FUNCTION_BLOCK FB_MotionAxis_MC

VAR_INPUT
	ZSN	   			: BOOL												;
	ZSP				: BOOL												; 
	Exceeding_us			: INT;
	sNameAxis				: STRING [40];

END_VAR         	
                	
VAR  
	rtFirstCycle	: R_TRIG;						
	mcHomeAxis		: 	MC_HomeAxis						;//ADD BY EVAN 
	sAxisName		: STRING											;//Axis name          	
	xPlus			: BOOL												;	
	xMinus			: BOOL												;
	bDone			: BOOL												;	

// Variables for Hard Stop Homing	                        			
	iStatehsHomig	: E_HomingSteps := E_HomingSteps.IDLE				;
	rtHome			: R_TRIG											;
	rtHomeReset		: R_TRIG											;
	tonTimeOut		: TON												;
	xTimerStart		: BOOL												;
	bLSDefaultVal	: BOOL												; // Save Def value from driver
	xHomeError		: BOOL												;
// Variables for Force Control          					

	rtForceC		: R_TRIG											;
	rtForceCReset	: R_TRIG											;
	DelMaxPos		: LREAL 											;
	rCurrLimit		: LREAL												;
	StartPos		: LREAL												;
	xForceCError	: BOOL												;
//	Variables for Backlash Compensation
	rLastMove		: LREAL := 1										;
	tonBackComp		: TON												;
	rBacklashPer	: LREAL												;	
	
// Variables for errors
	rtError					:	R_TRIG;
	pTextType				:	POINTER TO STRING;
	sAxisErrorID			:	STRING(10);	
	ErrorMSG				:	STRING[255];

//	Exceeding time measuring
	sysTime					:	GETCPUCOUNTER;//GETSYSTEMTIME;					//	Used to measure execution time.
	uStartTime				:	UDINT;
	uFinishTime				:	UDINT;
	ftimeDiff				:	REAL;
	ton_dly	: TON;
	offset	: WORD;
END_VAR         	
                	
VAR_IN_OUT      	
	IN_OUT 			: ST_MotionAxis_MC	;//struct for each axis
	AXIS 			: AXIS_REF			;//Axis obj	
END_VAR

VAR_OUTPUT
	xError			: BOOL				;
	xBusy			: BOOL				;
END_VAR
VAR CONSTANT
	parallelGroupTLName		:	STRING := 'Port_851.TL_Axis_Error';
END_VAR

(* Power options ********************************************************************************************)			
IN_OUT.mcPower(
	Axis				:= AXIS, 
	Enable				:= , 
	Enable_Positive		:= ZSP, 
	Enable_Negative		:= ZSN OR IN_OUT.mcHome.Busy, 
	Override			:= , 
	BufferMode			:= , 
	Options				:= , 
	Status				=> , 
	Busy				=> , 
	Active				=> , 
	Error				=> , 
	ErrorID				=> );
	
(* Halt Mode ********************************************************************************************)	
IN_OUT.mcHalt(
	Axis				:= AXIS, 
	Execute				:= , 
	Deceleration		:= IN_OUT.rDeceleration, 
	Jerk				:= , 
	BufferMode			:= , 
	Options				:= , 
	Done				=> , 
	Busy				=> , 
	Active				=> , 
	CommandAborted		=> , 
	Error				=> , 
	ErrorID				=> );
	
(* Homing ***********************************************************************************************)
IN_OUT.mcHome(
	Axis				:= AXIS, 
	Execute				:= , 
	Position			:= in_out.rFirstpos, 
	HomingMode			:= MC_Direct, 
	BufferMode			:= , 
	Options				:= , 
	bCalibrationCam		:= ,//NOT  ZSN, 
	Done				=> , 
	Busy				=> , 
	Active				=> , 
	CommandAborted		=> , 
	Error				=> , 
	ErrorID				=> );
	
(* JOG **************************************************************************************************)
IN_OUT.mcJog(
	Axis				:= AXIS, 
	JogForward			:= , 
	JogBackwards		:= , 
	Mode				:= E_JogMode.MC_JOGMODE_CONTINOUS, 
	Position			:= , 
	Velocity			:= IN_OUT.rVelocity, 
	Acceleration		:= IN_OUT.rAcceleration, 
	Deceleration		:= IN_OUT.rDeceleration, 
	Jerk				:= IN_OUT.rJerk, 
	Done				=> , 
	Busy				=> , 
	Active				=> , 
	CommandAborted		=> , 
	Error				=> , 
	ErrorID				=> );
	
(* Move Absolute ****************************************************************************************)	
IN_OUT.mcMoveAbsolute(
	Axis				:= AXIS, 
	Execute				:= , 
	Position			:= IN_OUT.rActualPosSet, 
	Velocity			:= IN_OUT.rVelocitySet,     
	Acceleration		:= IN_OUT.rAcceleration, 
	Deceleration		:= IN_OUT.rDeceleration, 
	Jerk				:= IN_OUT.rJerk,         
	BufferMode			:= , 
	Options				:= , 
	Done				=> , 
	Busy				=> , 
	Active				=> , 
	CommandAborted		=> , 
	Error				=> , 
	ErrorID				=> );

	IF IN_OUT.bMoveAbsHMI THEN
		IN_OUT.mcMoveAbsolute.Execute	:= TRUE;
		IN_OUT.rActualPosSet	:= IN_OUT.rActualPosHMI;
		IN_OUT.rVelocitySet		:= IN_OUT.rVeloPers;
	END_IF
(* Move Relative *********************************************************************************************************)
IN_OUT.mcMoveRelative(
	Axis				:= AXIS, 
	Execute				:= , 
	Distance			:= IN_OUT.rPosition + IN_OUT.rBacklashvalue, 
	Velocity			:= IN_OUT.rVelocity,      
	Acceleration		:= IN_OUT.rAcceleration,  
	Deceleration		:= IN_OUT.rDeceleration,  
	Jerk				:= IN_OUT.rJerk,          
	BufferMode			:= ,
	Options				:= , 
	Done				=> bDone, 
	Busy				=> , 
	Active				=> , 
	CommandAborted		=> , 
	Error				=> , 
	ErrorID				=> );
	
(* Move Velocity *********************************************************************************************************)
	
IN_OUT.mcMoveVelocity(
	Axis				:=	AXIS,
	Execute				:=	,
	Velocity			:=	IN_OUT.rVelocity,
	Acceleration		:=	IN_OUT.rAcceleration,
	Deceleration		:=	IN_OUT.rDeceleration,
	Jerk				:=	IN_OUT.rJerk,
	Direction			:=	IN_OUT.axisDirection,
	BufferMode			:=	,
	Options				:=	,
	InVelocity			=>	,
	Busy				=>	,
	Active				=>	,
	CommandAborted		=>	,
	Error				=>	,
	ErrorID				=>	);
	
(**)	
IN_OUT.mcReadStatus(
	Axis				:= AXIS, 
	Enable				:= TRUE, 
	Valid				=> , 
	Busy				=> , 
	Error				=> , 
	ErrorID				=> , 
	ErrorStop			=> , 
	Disabled			=> , 
	Stopping			=> , 
	StandStill			=> , 
	DiscreteMotion		=> , 
	ContinuousMotion	=> , 
	SynchronizedMotion	=> , 
	Homing				=> , 
	ConstantVelocity	=> , 
	Accelerating		=> , 
	Decelerating		=> , 
	Status				=> );
	
(* Reset ************************************************************************************************)
IN_OUT.mcReset(
	Axis				:= AXIS, 
	Execute				:= , 
	Done				=> , 
	Busy				=> , 
	Error				=> , 
	ErrorID				=> );
	
(* Stop *************************************************************************************************)
IN_OUT.mcStop(
	Axis				:= AXIS, 
	Execute				:= , 
	Deceleration		:= , 
	Jerk				:= , 
	Options				:= , 
	Done				=> , 
	Busy				=> , 
	Active				=> , 
	CommandAborted		=> , 
	Error				=> , 
	ErrorID				=> );

(* Set Position *************************************************************************************************)
in_out.mcSetpoint(
	Axis			 := AXIS, 
	Execute			 := , 
	Position		 := IN_OUT.rSetPos, 
	Mode			 := , 
	Options			 := , 
	Done			 => , 
	Busy			 => , 
	Error			 => , 
	ErrorID			 => );


(* write status *************************************************************************************************)
IN_OUT.mcWriteBoolParameter(
	Axis			:= 	AXIS, 
	Execute:= 				, 
	ParameterNumber:= 		, 
	Value:= , 
	Done=> , 
	Busy=> , 
	Error=> , 
	ErrorID=> );

(* Read status *************************************************************************************************)
IN_OUT.mcReadBoolParameter(
	Axis:= AXIS, 
	Enable:= , 
	ParameterNumber:= , 
	ReadMode:= , 
	Valid=> , 
	Busy=> , 
	Error=> , 
	ErrorID=> , 
	Value=> );	

(*Read Actualposition***************************************************************)
IN_OUT.mcReadActualPosition(
	Axis:= AXIS, 
	Enable:= TRUE, 
	Valid=> , 
	Busy=> , 
	Error=> , 
	ErrorID=> , 
	Position=> IN_OUT.rActualPos );   
(*COE write**************************************************************************)	

IN_OUT.CoeWrt(
	sNetId:= IN_OUT.sNetID, 
	nSlaveAddr:= IN_OUT.nSlaveAddr, 
	nSubIndex:= IN_OUT.nSubIndex, 
	nIndex:= IN_OUT.nIndex, 
	pSrcBuf:= ADR(IN_OUT.iSdoWrite), 
	cbBufLen:= SIZEOF(IN_OUT.iSdoWrite), 
	bExecute:= , 
	tTimeout:= , 
	bBusy=> , 
	bError=> , 
	nErrId=> );
	ton_dly(PT:=T#100MS);


offset	:= 16#800*IN_OUT.iAxis;	
CASE IN_OUT.iCoeWrt OF 
	0:
		IN_OUT.CoeWrt.bExecute := FALSE;
	1:
		IN_OUT.CoeWrt.bExecute := TRUE;
		IN_OUT.nIndex	:= 16#2005+offset;
		IN_OUT.nSubIndex	:= 16#1F;
		IN_OUT.iSdoWrite	:= 6;//clear encoder and set current position as origin
		IN_OUT.iCoeWrt	:= 10;
	2:
		IN_OUT.CoeWrt.bExecute := TRUE;
		IN_OUT.nIndex	:= 16#2002+offset;
		IN_OUT.nSubIndex	:= 16#02;
		IN_OUT.iSdoWrite	:= 1;//linear mode
		IN_OUT.iCoeWrt	:= 10;
	3:
		IN_OUT.CoeWrt.bExecute := TRUE;
		IN_OUT.nIndex	:= 16#2002+offset;
		IN_OUT.nSubIndex	:= 16#02;
		IN_OUT.iSdoWrite	:= 2;//rotate mode
		IN_OUT.iCoeWrt	:= 10;
	4:
		IN_OUT.CoeWrt.bExecute := TRUE;
		IN_OUT.nIndex	:= 16#2004+offset;
		IN_OUT.nSubIndex	:= 16#06;
		IN_OUT.iSdoWrite	:= 1;//breaker on
		IN_OUT.iCoeWrt	:= 10;
	5:
		IN_OUT.CoeWrt.bExecute := TRUE;
		IN_OUT.nIndex	:= 16#2004+offset;
		IN_OUT.nSubIndex	:= 16#06;
		IN_OUT.iSdoWrite	:= 0;//breaker off
		IN_OUT.iCoeWrt	:= 10;		
	10:		
		IN_OUT.iCoeWrt	:= 0;
END_CASE







	(*mcHomeAxis***************************************************************)
	mcHomeAxis(
		xExecute:= , 
		xReset:= , 
		InOut:=IN_OUT , 
		xRedy=> , 
		xBusy=> , 
		xDone=> , 
		xError=> ); 
	                                                                                                              	
(******************************************************************************************************************)
	
(**error flag**)

	IN_OUT.xTorqueErr	:=ABS(IN_OUT.rActTorque)>IN_OUT.rToqueLimitSet ;

	
	

	xError := IN_OUT.mcReadStatus.Error OR xHomeError OR IN_OUT.mcMoveAbsolute.Error OR IN_OUT.xTorqueErr ;	
	rtError(CLK:= (IN_OUT.mcReadStatus.ErrorID <> 0 OR xError) AND NOT IN_OUT.xMuteAxisErrorMessages);
	
(*************************** READ ERROR FROM DRIVE *************************)
rtFirstCycle(CLK:= TRUE);
sysTime(cpuCntLoDW => uStartTime);	
sysTime(cpuCntLoDW => uFinishTime);
//M_CheckExceedingTime();

(*************************** GET AXIS ERROR MESSAGE *************************)	
	
	IF rtError.Q THEN
		IF IN_OUT.xTorqueErr THEN
			sAxisErrorID	:= 'TORQUE';
		ELSE
			sAxisErrorID	:=	TO_STRING(IN_OUT.mcReadStatus.ErrorID);
		END_IF
		IN_OUT.mcStop.Execute	:= TRUE;
	
	END_IF
(**remember the Velocity**) 
	IF IN_OUT.rVeloPers <> 0 THEN 
		IN_OUT.rVelocity:= IN_OUT.rVeloPers;
	ELSE 
		IN_OUT.rVeloPers := IN_OUT.rVelocity;	
	END_IF	
(**remember the Acceleration**)
	IF IN_OUT.rAccPers <> 0 THEN 
		IN_OUT.rAcceleration:= IN_OUT.rAccPers;
	ELSE 
		IN_OUT.rAccPers := IN_OUT.rAcceleration;		
	END_IF	
(**remember the Deceleration**)
	IF IN_OUT.rDecPers <> 0 THEN 
		IN_OUT.rDeceleration:= IN_OUT.rDecPers;
	ELSE 
		IN_OUT.rDecPers := IN_OUT.rDeceleration;		
	END_IF
(**False all Executions if function done or error**)
	IF IN_OUT.mcMoveRelative.Done OR IN_OUT.mcMoveRelative.Error OR IN_OUT.mcReset.Busy THEN 
		IN_OUT.mcMoveRelative.Execute := FALSE;
	END_IF

	IF IN_OUT.mcMoveVelocity.Error OR IN_OUT.mcReset.Busy OR IN_OUT.mcMoveVelocity.Busy THEN 
		IN_OUT.mcMoveVelocity.Execute := FALSE;
	END_IF
	
	IF IN_OUT.mcSetpoint.done OR IN_OUT.mcSetpoint.Error THEN
		IN_OUT.mcSetpoint.Execute := FALSE;
	END_IF
	
    IF  IN_OUT.mcMoveAbsolute.Done OR IN_OUT.mcMoveAbsolute.Error OR IN_OUT.mcReset.Busy THEN 
		IN_OUT.mcMoveAbsolute.Execute := FALSE;
	END_IF
 
	 IF IN_OUT.mcHome.Done OR IN_OUT.mcHome.Error THEN 
		IN_OUT.mcHome.Execute := FALSE;
	END_IF
	
	IF IN_OUT.mcStop.Done OR IN_OUT.mcStop.Error THEN 
		IN_OUT.mcStop.Execute := FALSE;
	END_IF
	
	IF IN_OUT.mcReset.Done OR IN_OUT.mcReset.Error THEN 
		IN_OUT.mcReset.Execute := FALSE;
	END_IF
			
	IF IN_OUT.mcReadBoolParameter.Valid OR IN_OUT.mcReadBoolParameter.Error THEN 
		IN_OUT.mcReadBoolParameter.Enable := FALSE;
	END_IF	
	
	IF IN_OUT.mcWriteBoolParameter.Done OR IN_OUT.mcWriteBoolParameter.Error THEN 
		IN_OUT.mcWriteBoolParameter.Execute	:= FALSE;
	END_IF	
		

	
	
	
(**Save done state into temp variable**)	
	
	IF IN_OUT.mcMoveAbsolute.Done THEN
		IN_OUT.xMoveABSDone := TRUE;
	END_IF	
	
	IF IN_OUT.mcMoveRelative.Done THEN
		IN_OUT.xMoveRelDone := TRUE;
	END_IF

PROPERTY P_AxisName : STRING
SET
sAxisName := P_AxisName;
END_SET
END_PROPERTY

PROPERTY P_CurrLimit : LREAL
SET
rCurrLimit := P_CurrLimit;
END_SET
END_PROPERTY

PROPERTY P_DelMaxPos : LREAL
SET
DelMaxPos := P_DelMaxPos;
END_SET
END_PROPERTY

PROPERTY P_ForceCError : BOOL
GET
P_ForceCError := xForceCError;
END_GET
END_PROPERTY

PROPERTY P_hsHomingError : BOOL
GET
P_hsHomingError := xHomeError;
END_GET
END_PROPERTY

PROPERTY P_StartPos : LREAL
SET
StartPos := P_StartPos;
END_SET
END_PROPERTY

END_FUNCTION_BLOCK

(* stored: Version 1.1.0.1, ProductVersion 3.1.4024.12
   POU FB_MotionAxis_MC: Id {ca80f1ef-324b-44ba-b9f2-eaf2b6169801}, SpecialFunc None
   Property P_AxisName: Id {094743f5-b136-48b4-b605-5fd26680bfed}
   Set Set: Id {2ccdb01d-0165-4d88-87b4-c11727f2bbff}
   Property P_CurrLimit: Id {519602c4-14a7-4327-a3ca-2f41ff6c5c5d}
   Set Set: Id {646e0e60-ec1e-4ace-bd79-1147f5e2df19}
   Property P_DelMaxPos: Id {6ecdb536-135e-42ba-b965-10bfd06a7473}
   Set Set: Id {b74d0b50-c12e-4360-9b39-447e2609d444}
   Property P_ForceCError: Id {c2c42c29-befb-4e3f-8671-2d2595f70133}
   Get Get: Id {22cd7458-0f90-4520-a424-7a3869e02703}
   Property P_hsHomingError: Id {74f2954d-cc04-4af4-95ab-3055da4fc7fc}
   Get Get: Id {5e238761-9ba9-4394-adc9-048eb9416b36}
   Property P_StartPos: Id {418ac9b2-b307-4f60-9c96-04382ba77b16}
   Set Set: Id {1c3ccce8-6631-457a-be08-e5f56bf41e9c} *)
